FUNCTION_BLOCK FB_ButtonBox
VAR_INPUT
	IN			: BOOL;
	State : 	(NOT_READY, ALL_READY, RUNNING, STOP, ERROR);	//Local ENUM
	Button1		: BOOL;
	SwitchLeft 	: BOOL;
	SwitchRight : BOOL;
END_VAR
VAR_OUTPUT
	Q 		: BOOL;
	RUN		: BOOL;
	oLight1 : BOOL;	
	Forward 	: BOOL;
	Backward 	: BOOL;
END_VAR
VAR
	BTN_Feed_TRIG: BOOL;
	Rtrig2: R_TRIG;
	Rtrig3: R_TRIG;
	tempCount1: INT;
	tempCount2: INT;
	tempCount3: INT;
	tempCount0: INT;

	RS1: RS;
	SwitchLeftRight_RS: BOOL;
	rTrig1: R_TRIG;
	RS_2: RS;
END_VAR

Q := IN;

// Button press handling
A_InputHandling();

// Button box light controls dictated by the state of Belt Control.
CASE State OF		// State is an input of 1-5 from BeltControl FB
	
	NOT_READY:
		oLight1 := FALSE;

	ALL_READY:
		oLight1 := GENERAL.BlinkOn;
		
	RUNNING:
		oLight1 := TRUE;		
		
	STOP:
		oLight1 := GENERAL.BlinkSpecial_On;

	ERROR:
		oLight1 := GENERAL.BlinkSpecial_On;
		
END_CASE

ACTION A_InputHandling:
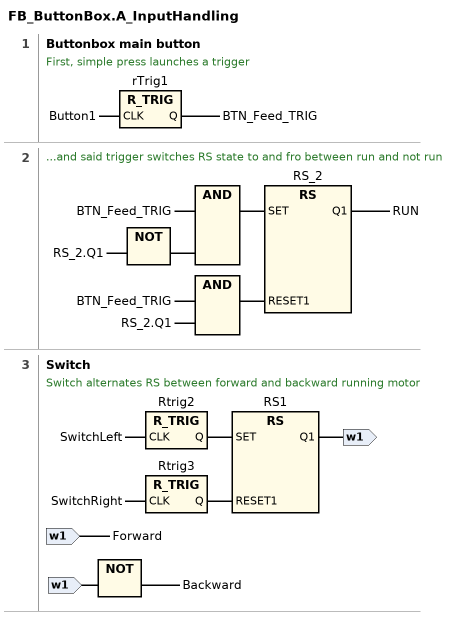
// NETWORK 1: Buttonbox main button
// First, simple press launches a trigger
rTrig1(CLK := Button1); // R_TRIG
BTN_Feed_TRIG := rTrig1.Q;

// NETWORK 2
// ...and said trigger switches RS state to and fro between run and not run
RS_2(SET := BTN_Feed_TRIG AND NOT RS_2.Q1, RESET1 := BTN_Feed_TRIG AND RS_2.Q1); // RS
RUN := RS_2.Q1;

// NETWORK 3: Switch
// Switch alternates RS between forward and backward running motor
Rtrig2(CLK := SwitchLeft); // R_TRIG
Rtrig3(CLK := SwitchRight); // R_TRIG
RS1(SET := Rtrig2.Q, RESET1 := Rtrig3.Q); // RS
Forward := RS1.Q1;
Backward := NOT RS1.Q1;
END_ACTION

END_FUNCTION_BLOCK

(* stored: Version 1.1.0.1, ProductVersion 3.1.4024.10
   POU FB_ButtonBox: Id {718ab21c-a86f-42b1-ad84-7eea86241524}, SpecialFunc None
   Action A_InputHandling: Id {3b6590fa-f99a-41e5-8828-c964d473a0f6} *)
